Fanuc KAREL source: ks00042.KL

-- PROVISIONAL review KL for V1013-1; original PC SHA256 bc2ea042ce332d2c29518f76c5d97e3cc0fdda34b59ff38c0354bdffa1e6134b
-- Incomplete behavior may be omitted. Consult companion uncertainty JSON. Do not deploy.
PROGRAM KS00042
%NOLOCKGROUP
BEGIN
  -- UNRESOLVED_PC offsets 5-13; opcodes 3F,75
  -- UNRESOLVED_PC offsets 18-27; opcodes 3F,75
  -- UNRESOLVED_PC offsets 32-70; opcodes 27,22,22,2A,22,2A,22,22,B0
  -- UNRESOLVED_PC offsets 75-79; opcodes 7F
END KS00042
